// TIA Portal V19 export
DATA_BLOCK "Main_Safety_RTG1_DB"   // DB166, F_DB
NAME : FUSI
// stored: InstanceOfName Main_Safety_RTG1, InstanceOfType FB
"Main_Safety_RTG1"
   // VAR
   //    ACK_GL : ACK_GL;
   //    F_Estop : "F_Estop_FB";
   //    F_Bimanuals : "F_TwoHands_FB";
   //    F_Zone00 : "F_Zone00_FB";
   //    F_Zone01_02_03 : "F_Zone01_02_03_FB";
   //    F_Zone05 : "F_Zone05_FB";
   //    F_Zone10 : "F_Zone10_FB";
   //    F_Zone11 : "F_Zone11_FB";
   //    F_Zone13 : "F_Zone13_FB";
   //    F_Zone15 : "F_Zone15_FB";
   //    F_Zone20 : "F_Zone20_FB";
   //    F_Zone21 : "F_Zone21_FB";
   //    F_Zone23 : "F_Zone23_FB";
   //    F_Zone25 : "F_Zone25_FB";
   //    F_Zone27 : "F_Zone27_FB";
   //    F_Zone29 : "F_Zone29_FB";
   // END_VAR
BEGIN
END_DATA_BLOCK
